{attribute 'no-analysis'}
FUNCTION_BLOCK StepManagerBasic_Test EXTENDS FB_TestSuite
VAR_INPUT
END_VAR
VAR_OUTPUT
END_VAR
VAR
END_VAR

// Copyright (c) 2024 Loupe (https://loupe.team), provided under the MIT License.

RequestStep();
Reset();

METHOD RequestStep
VAR
    stepManager : StepManagerBasic();
END_VAR
// Copyright (c) 2024 Loupe (https://loupe.team), provided under the MIT License.

(*STweep.Disable*)

TEST('RequestStep');
	stepManager.RequestStep(2);
	AssertEquals_UDINT(Expected := 2, Actual := stepManager.currentStep, 'Current Step shall be requested step');
TEST_FINISHED();
END_METHOD

METHOD Reset
VAR
    stepManager : StepManagerBasic();
END_VAR
// Copyright (c) 2024 Loupe (https://loupe.team), provided under the MIT License.

(*STweep.Disable*)

TEST('Reset');
	stepManager.RequestStep(20);
	AssertEquals_UDINT(Expected := 20, Actual := stepManager.currentStep, 'Confirm current step is not default');
	
	stepManager.Reset();
	AssertEquals_UDINT(Expected := SEQUENCE_STEP.NO_STEP, Actual := stepManager.currentStep, 'Reset should have put current step back to default');
TEST_FINISHED();
END_METHOD

END_FUNCTION_BLOCK

(* stored: Version 1.1.0.1
   POU StepManagerBasic_Test: Id {f2f4fe9e-d358-482a-b327-02ec29657bd0}, SpecialFunc None
   Method RequestStep: Id {198c2120-5857-4c31-b6b8-c5eeca56d028}
   Method Reset: Id {f87175cc-f817-48db-aeb6-5cea267ae2ed} *)
